PROGRAM MAIN
VAR
	Estacion: FB_Estacion;
END_VAR

Estacion();

END_PROGRAM

(* stored: Version 1.1.0.1, ProductVersion 3.1.4024.12
   POU MAIN: Id {6534206c-4aed-4051-b454-4515e10637f3}, SpecialFunc None *)
